FUNCTION_BLOCK FB_SimpleLog
VAR_INPUT
	Message: 		STRING(255) := '';
END_VAR
VAR_OUTPUT
END_VAR
VAR
	// ADSLOG_MSGTYPE_HINT or ADSLOG_MSGTYPE_WARN or ADSLOG_MSGTYPE_ERROR
	Level:			UDINT := ADSLOG_MSGTYPE_HINT;
	FormatString: 	STRING(255) := '%s';
	LastMessage:		STRING(255) := '';
END_VAR

IF Message <> LastMessage THEN
	ADSLOGSTR( Level OR ADSLOG_MSGTYPE_LOG, FormatString, Message);
END_IF
LastMessage := Message;

END_FUNCTION_BLOCK

(* stored: Version 1.1.0.1, ProductVersion 3.1.4024.6
   POU FB_SimpleLog: Id {a26a3b36-e872-4925-b825-b15d2b0093fa}, SpecialFunc None *)
